// TIA Portal V16 export
// export: Created 2022-09-01T14:26:54.6640188Z, ExportSetting WithDefaults, DisplayName Totally Integrated Automation Portal, DisplayVersion V16, DisplayName TIA Portal Version Control Interface, DisplayVersion V16, DisplayName TIA Portal Openness, DisplayVersion V16, DisplayName STEP 7 Professional, DisplayVersion V16, DisplayName STEP 7 Safety, DisplayVersion V16, DisplayName WinCC Advanced, DisplayVersion V16
FUNCTION "Saídas_Bombas" : Void   // FC3, LAD
{ S7_Optimized_Access := 'TRUE' }
VERSION : 0.1
// stored: AutoNumber true, IsIECCheckEnabled false, SetENOAutomatically false, UDAEnableTagReadback false
   VAR_TEMP
      BOMBA_1_VAR : Bool;
      BOMBA_2_VAR : Bool;
      BOMBA_3_RESERVA : Bool;
   END_VAR
BEGIN

REGION Network 1: Bomba 1 (com variador)
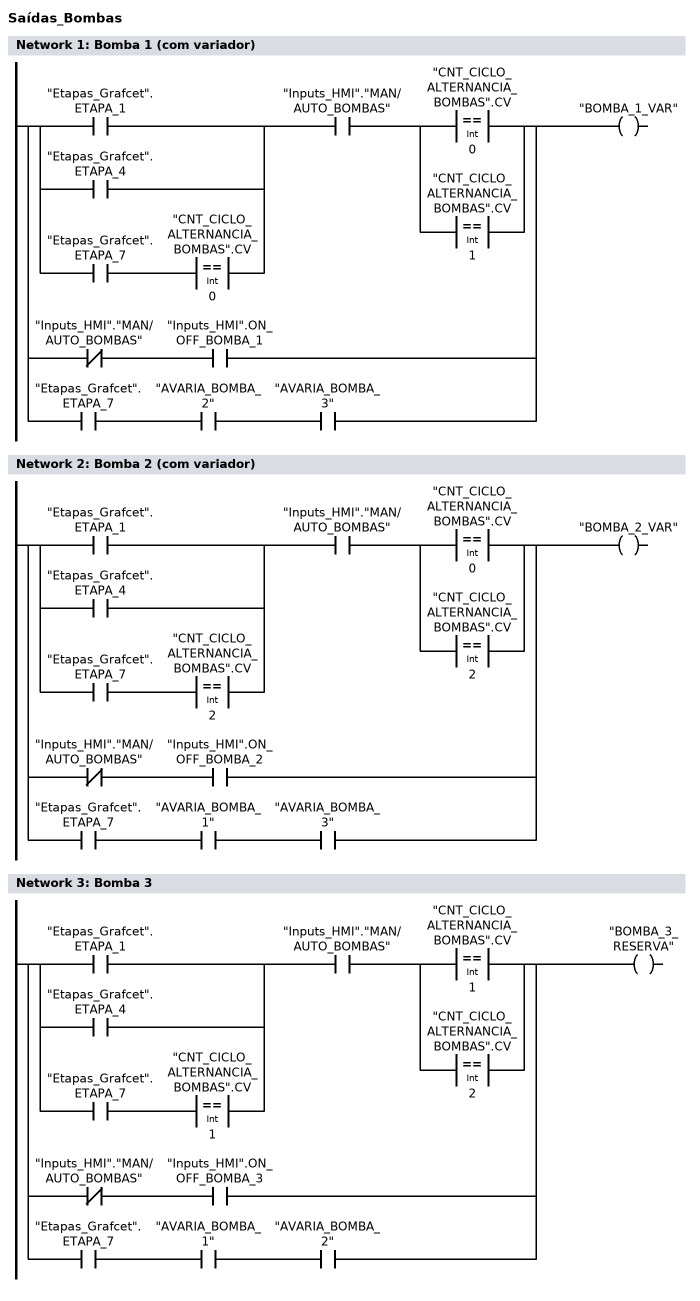
   RUNG wire#powerrail
      Contact( "Etapas_Grafcet".ETAPA_1 )
      wire#w1
      Contact( "Inputs_HMI"."MAN/AUTO_BOMBAS" )
      wire#w2
      { S7_Templates := "SrcType := Int" } EQ_Contact(in1 := "CNT_CICLO_ALTERNANCIA_BOMBAS".CV, in2 := 0)
      wire#w3
      Coil( "BOMBA_1_VAR" )
   END_RUNG
   RUNG wire#powerrail
      Contact( "Etapas_Grafcet".ETAPA_4 )
   END_RUNG wire#w1
   RUNG wire#powerrail
      Contact( "Etapas_Grafcet".ETAPA_7 )
      { S7_Templates := "SrcType := Int" } EQ_Contact(in1 := "CNT_CICLO_ALTERNANCIA_BOMBAS".CV, in2 := 0)
   END_RUNG wire#w1
   RUNG wire#w2
      { S7_Templates := "SrcType := Int" } EQ_Contact(in1 := "CNT_CICLO_ALTERNANCIA_BOMBAS".CV, in2 := 1)
   END_RUNG wire#w3
   RUNG wire#powerrail
      I_Contact( "Inputs_HMI"."MAN/AUTO_BOMBAS" )
      Contact( "Inputs_HMI".ON_OFF_BOMBA_1 )
   END_RUNG wire#w3
   RUNG wire#powerrail
      Contact( "Etapas_Grafcet".ETAPA_7 )
      Contact( "AVARIA_BOMBA_2" )
      Contact( "AVARIA_BOMBA_3" )
   END_RUNG wire#w3
   // the same network as SCL:
   "BOMBA_1_VAR" := (("Etapas_Grafcet".ETAPA_1 OR "Etapas_Grafcet".ETAPA_4 OR ("Etapas_Grafcet".ETAPA_7 AND ("CNT_CICLO_ALTERNANCIA_BOMBAS".CV = 0))) AND "Inputs_HMI"."MAN/AUTO_BOMBAS" AND (("CNT_CICLO_ALTERNANCIA_BOMBAS".CV = 0) OR ("CNT_CICLO_ALTERNANCIA_BOMBAS".CV = 1))) OR (NOT "Inputs_HMI"."MAN/AUTO_BOMBAS" AND "Inputs_HMI".ON_OFF_BOMBA_1) OR ("Etapas_Grafcet".ETAPA_7 AND "AVARIA_BOMBA_2" AND "AVARIA_BOMBA_3");
END_REGION

REGION Network 2: Bomba 2 (com variador)
   RUNG wire#powerrail
      Contact( "Etapas_Grafcet".ETAPA_1 )
      wire#w1
      Contact( "Inputs_HMI"."MAN/AUTO_BOMBAS" )
      wire#w2
      { S7_Templates := "SrcType := Int" } EQ_Contact(in1 := "CNT_CICLO_ALTERNANCIA_BOMBAS".CV, in2 := 0)
      wire#w3
      Coil( "BOMBA_2_VAR" )
   END_RUNG
   RUNG wire#powerrail
      Contact( "Etapas_Grafcet".ETAPA_4 )
   END_RUNG wire#w1
   RUNG wire#powerrail
      Contact( "Etapas_Grafcet".ETAPA_7 )
      { S7_Templates := "SrcType := Int" } EQ_Contact(in1 := "CNT_CICLO_ALTERNANCIA_BOMBAS".CV, in2 := 2)
   END_RUNG wire#w1
   RUNG wire#w2
      { S7_Templates := "SrcType := Int" } EQ_Contact(in1 := "CNT_CICLO_ALTERNANCIA_BOMBAS".CV, in2 := 2)
   END_RUNG wire#w3
   RUNG wire#powerrail
      I_Contact( "Inputs_HMI"."MAN/AUTO_BOMBAS" )
      Contact( "Inputs_HMI".ON_OFF_BOMBA_2 )
   END_RUNG wire#w3
   RUNG wire#powerrail
      Contact( "Etapas_Grafcet".ETAPA_7 )
      Contact( "AVARIA_BOMBA_1" )
      Contact( "AVARIA_BOMBA_3" )
   END_RUNG wire#w3
   // the same network as SCL:
   "BOMBA_2_VAR" := (("Etapas_Grafcet".ETAPA_1 OR "Etapas_Grafcet".ETAPA_4 OR ("Etapas_Grafcet".ETAPA_7 AND ("CNT_CICLO_ALTERNANCIA_BOMBAS".CV = 2))) AND "Inputs_HMI"."MAN/AUTO_BOMBAS" AND (("CNT_CICLO_ALTERNANCIA_BOMBAS".CV = 0) OR ("CNT_CICLO_ALTERNANCIA_BOMBAS".CV = 2))) OR (NOT "Inputs_HMI"."MAN/AUTO_BOMBAS" AND "Inputs_HMI".ON_OFF_BOMBA_2) OR ("Etapas_Grafcet".ETAPA_7 AND "AVARIA_BOMBA_1" AND "AVARIA_BOMBA_3");
END_REGION

REGION Network 3: Bomba 3
   RUNG wire#powerrail
      Contact( "Etapas_Grafcet".ETAPA_1 )
      wire#w1
      Contact( "Inputs_HMI"."MAN/AUTO_BOMBAS" )
      wire#w2
      { S7_Templates := "SrcType := Int" } EQ_Contact(in1 := "CNT_CICLO_ALTERNANCIA_BOMBAS".CV, in2 := 1)
      wire#w3
      Coil( "BOMBA_3_RESERVA" )
   END_RUNG
   RUNG wire#powerrail
      Contact( "Etapas_Grafcet".ETAPA_4 )
   END_RUNG wire#w1
   RUNG wire#powerrail
      Contact( "Etapas_Grafcet".ETAPA_7 )
      { S7_Templates := "SrcType := Int" } EQ_Contact(in1 := "CNT_CICLO_ALTERNANCIA_BOMBAS".CV, in2 := 1)
   END_RUNG wire#w1
   RUNG wire#w2
      { S7_Templates := "SrcType := Int" } EQ_Contact(in1 := "CNT_CICLO_ALTERNANCIA_BOMBAS".CV, in2 := 2)
   END_RUNG wire#w3
   RUNG wire#powerrail
      I_Contact( "Inputs_HMI"."MAN/AUTO_BOMBAS" )
      Contact( "Inputs_HMI".ON_OFF_BOMBA_3 )
   END_RUNG wire#w3
   RUNG wire#powerrail
      Contact( "Etapas_Grafcet".ETAPA_7 )
      Contact( "AVARIA_BOMBA_1" )
      Contact( "AVARIA_BOMBA_2" )
   END_RUNG wire#w3
   // the same network as SCL:
   "BOMBA_3_RESERVA" := (("Etapas_Grafcet".ETAPA_1 OR "Etapas_Grafcet".ETAPA_4 OR ("Etapas_Grafcet".ETAPA_7 AND ("CNT_CICLO_ALTERNANCIA_BOMBAS".CV = 1))) AND "Inputs_HMI"."MAN/AUTO_BOMBAS" AND (("CNT_CICLO_ALTERNANCIA_BOMBAS".CV = 1) OR ("CNT_CICLO_ALTERNANCIA_BOMBAS".CV = 2))) OR (NOT "Inputs_HMI"."MAN/AUTO_BOMBAS" AND "Inputs_HMI".ON_OFF_BOMBA_3) OR ("Etapas_Grafcet".ETAPA_7 AND "AVARIA_BOMBA_1" AND "AVARIA_BOMBA_2");
END_REGION
END_FUNCTION
